// TIA Portal V19 export
FUNCTION "CollectAlarms" : Void   // FC58, LAD
TITLE = Alarm Collector Equipment
// Collects alarms from the respective level and categorises the alarms into the different alarm classes. Filling the alarm DB with specific alarm messages which are defined in the comment of the defined alarm. The definition of possible alarms within a equipment is handled here.
// stored: IsIECCheckEnabled true, Namespace Unit.Em2, SetENOAutomatically true
   VAR_INPUT
      resetAlarms : Bool;   // Reset the currently pending alarms
      disableAlarms : Bool;   // Disable all the Alarms - pending alarms will stay until a reset is triggered
   END_VAR
   VAR_OUTPUT
      commandsToUnit : "LUC_typeStateCommands";   // Feedback to the unit
   END_VAR
BEGIN

REGION Network 1: Reset Alarms
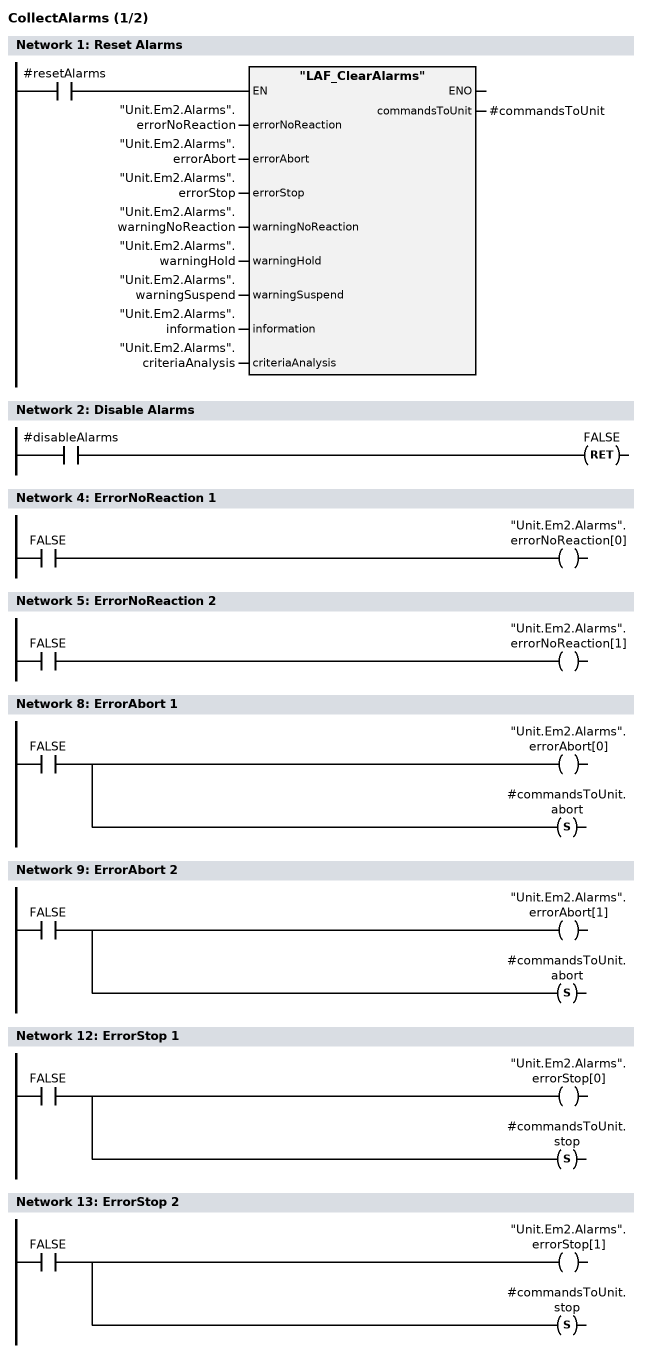
   RUNG wire#powerrail
      Contact( #resetAlarms )
      "LAF_ClearAlarms"(errorNoReaction := "Unit.Em2.Alarms".errorNoReaction, errorAbort := "Unit.Em2.Alarms".errorAbort, errorStop := "Unit.Em2.Alarms".errorStop, warningNoReaction := "Unit.Em2.Alarms".warningNoReaction, warningHold := "Unit.Em2.Alarms".warningHold, warningSuspend := "Unit.Em2.Alarms".warningSuspend, information := "Unit.Em2.Alarms".information, criteriaAnalysis := "Unit.Em2.Alarms".criteriaAnalysis, commandsToUnit => #commandsToUnit)
   END_RUNG
   // the same network as SCL:
   IF #resetAlarms THEN
       "LAF_ClearAlarms"(errorNoReaction := "Unit.Em2.Alarms".errorNoReaction,
                         errorAbort := "Unit.Em2.Alarms".errorAbort,
                         errorStop := "Unit.Em2.Alarms".errorStop,
                         warningNoReaction := "Unit.Em2.Alarms".warningNoReaction,
                         warningHold := "Unit.Em2.Alarms".warningHold,
                         warningSuspend := "Unit.Em2.Alarms".warningSuspend,
                         information := "Unit.Em2.Alarms".information,
                         criteriaAnalysis := "Unit.Em2.Alarms".criteriaAnalysis,
                         commandsToUnit => #commandsToUnit);
   END_IF;
END_REGION

REGION Network 2: Disable Alarms
   RUNG wire#powerrail
      Contact( #disableAlarms )
      ReturnCoil( FALSE )
   END_RUNG
   // the same network as SCL:
   IF #disableAlarms THEN
       ENO := FALSE;
       RETURN;
   END_IF;
END_REGION

REGION Network 3: *************** Error No Reaction ************************
END_REGION

REGION Network 4: ErrorNoReaction 1
   RUNG wire#powerrail
      Contact( FALSE )
      Coil( "Unit.Em2.Alarms".errorNoReaction[0] )
   END_RUNG
   // the same network as SCL:
   "Unit.Em2.Alarms".errorNoReaction[0] := FALSE;
END_REGION

REGION Network 5: ErrorNoReaction 2
   RUNG wire#powerrail
      Contact( FALSE )
      Coil( "Unit.Em2.Alarms".errorNoReaction[1] )
   END_RUNG
   // the same network as SCL:
   "Unit.Em2.Alarms".errorNoReaction[1] := FALSE;
END_REGION

REGION Network 7: *************** Error and Abort **************************
END_REGION

REGION Network 8: ErrorAbort 1
   RUNG wire#powerrail
      Contact( FALSE )
      wire#w1
      Coil( "Unit.Em2.Alarms".errorAbort[0] )
   END_RUNG
   RUNG wire#w1
      S_Coil( #commandsToUnit.abort )
   END_RUNG
   // the same network as SCL:
   "Unit.Em2.Alarms".errorAbort[0] := FALSE;
   IF FALSE THEN #commandsToUnit.abort := TRUE; END_IF;
END_REGION

REGION Network 9: ErrorAbort 2
   RUNG wire#powerrail
      Contact( FALSE )
      wire#w1
      Coil( "Unit.Em2.Alarms".errorAbort[1] )
   END_RUNG
   RUNG wire#w1
      S_Coil( #commandsToUnit.abort )
   END_RUNG
   // the same network as SCL:
   "Unit.Em2.Alarms".errorAbort[1] := FALSE;
   IF FALSE THEN #commandsToUnit.abort := TRUE; END_IF;
END_REGION

REGION Network 11: *************** Error and Stop ***************************
END_REGION

REGION Network 12: ErrorStop 1
   RUNG wire#powerrail
      Contact( FALSE )
      wire#w1
      Coil( "Unit.Em2.Alarms".errorStop[0] )
   END_RUNG
   RUNG wire#w1
      S_Coil( #commandsToUnit.stop )
   END_RUNG
   // the same network as SCL:
   "Unit.Em2.Alarms".errorStop[0] := FALSE;
   IF FALSE THEN #commandsToUnit.stop := TRUE; END_IF;
END_REGION

REGION Network 13: ErrorStop 2
   RUNG wire#powerrail
      Contact( FALSE )
      wire#w1
      Coil( "Unit.Em2.Alarms".errorStop[1] )
   END_RUNG
   RUNG wire#w1
      S_Coil( #commandsToUnit.stop )
   END_RUNG
   // the same network as SCL:
   "Unit.Em2.Alarms".errorStop[1] := FALSE;
   IF FALSE THEN #commandsToUnit.stop := TRUE; END_IF;
END_REGION

REGION Network 15: *************** Warning No Reaction **********************
END_REGION

REGION Network 16: WarningNoReaction 1
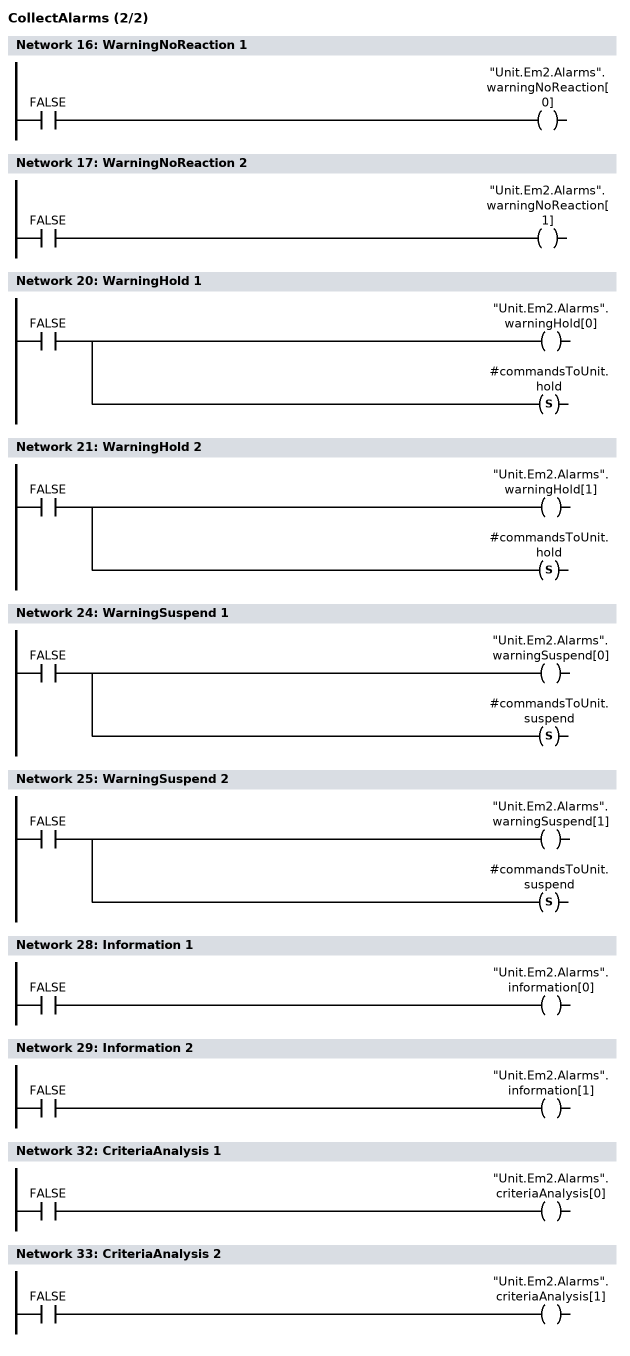
   RUNG wire#powerrail
      Contact( FALSE )
      Coil( "Unit.Em2.Alarms".warningNoReaction[0] )
   END_RUNG
   // the same network as SCL:
   "Unit.Em2.Alarms".warningNoReaction[0] := FALSE;
END_REGION

REGION Network 17: WarningNoReaction 2
   RUNG wire#powerrail
      Contact( FALSE )
      Coil( "Unit.Em2.Alarms".warningNoReaction[1] )
   END_RUNG
   // the same network as SCL:
   "Unit.Em2.Alarms".warningNoReaction[1] := FALSE;
END_REGION

REGION Network 19: *************** Warning Hold **************************
END_REGION

REGION Network 20: WarningHold 1
   RUNG wire#powerrail
      Contact( FALSE )
      wire#w1
      Coil( "Unit.Em2.Alarms".warningHold[0] )
   END_RUNG
   RUNG wire#w1
      S_Coil( #commandsToUnit.hold )
   END_RUNG
   // the same network as SCL:
   "Unit.Em2.Alarms".warningHold[0] := FALSE;
   IF FALSE THEN #commandsToUnit.hold := TRUE; END_IF;
END_REGION

REGION Network 21: WarningHold 2
   RUNG wire#powerrail
      Contact( FALSE )
      wire#w1
      Coil( "Unit.Em2.Alarms".warningHold[1] )
   END_RUNG
   RUNG wire#w1
      S_Coil( #commandsToUnit.hold )
   END_RUNG
   // the same network as SCL:
   "Unit.Em2.Alarms".warningHold[1] := FALSE;
   IF FALSE THEN #commandsToUnit.hold := TRUE; END_IF;
END_REGION

REGION Network 23: *************** Warning Suspend ***********************
END_REGION

REGION Network 24: WarningSuspend 1
   RUNG wire#powerrail
      Contact( FALSE )
      wire#w1
      Coil( "Unit.Em2.Alarms".warningSuspend[0] )
   END_RUNG
   RUNG wire#w1
      S_Coil( #commandsToUnit.suspend )
   END_RUNG
   // the same network as SCL:
   "Unit.Em2.Alarms".warningSuspend[0] := FALSE;
   IF FALSE THEN #commandsToUnit.suspend := TRUE; END_IF;
END_REGION

REGION Network 25: WarningSuspend 2
   RUNG wire#powerrail
      Contact( FALSE )
      wire#w1
      Coil( "Unit.Em2.Alarms".warningSuspend[1] )
   END_RUNG
   RUNG wire#w1
      S_Coil( #commandsToUnit.suspend )
   END_RUNG
   // the same network as SCL:
   "Unit.Em2.Alarms".warningSuspend[1] := FALSE;
   IF FALSE THEN #commandsToUnit.suspend := TRUE; END_IF;
END_REGION

REGION Network 27: *************** Information *****************************
END_REGION

REGION Network 28: Information 1
   RUNG wire#powerrail
      Contact( FALSE )
      Coil( "Unit.Em2.Alarms".information[0] )
   END_RUNG
   // the same network as SCL:
   "Unit.Em2.Alarms".information[0] := FALSE;
END_REGION

REGION Network 29: Information 2
   RUNG wire#powerrail
      Contact( FALSE )
      Coil( "Unit.Em2.Alarms".information[1] )
   END_RUNG
   // the same network as SCL:
   "Unit.Em2.Alarms".information[1] := FALSE;
END_REGION

REGION Network 31: *************** CriteriaAnalysis **************************
END_REGION

REGION Network 32: CriteriaAnalysis 1
   RUNG wire#powerrail
      Contact( FALSE )
      Coil( "Unit.Em2.Alarms".criteriaAnalysis[0] )
   END_RUNG
   // the same network as SCL:
   "Unit.Em2.Alarms".criteriaAnalysis[0] := FALSE;
END_REGION

REGION Network 33: CriteriaAnalysis 2
   RUNG wire#powerrail
      Contact( FALSE )
      Coil( "Unit.Em2.Alarms".criteriaAnalysis[1] )
   END_RUNG
   // the same network as SCL:
   "Unit.Em2.Alarms".criteriaAnalysis[1] := FALSE;
END_REGION
END_FUNCTION
